Yaskawa INFORM job: MALBEN4.JBI

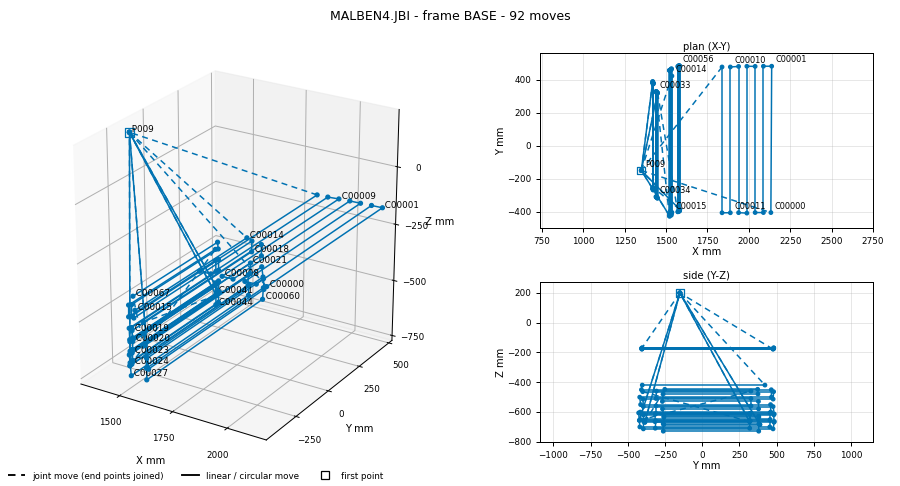
[picture p0: tool path of MALBEN4.JBI in frame BASE, 92 of 92 moves have a stored position in this frame; points joined in program order, loops and branches not executed]
/JOB
//NAME MALBEN4
//POS
///NPOS 86,0,86,1,0,1
///TOOL 0
///POSTYPE BASE
///RECTAN
///RCONF 1,0,0,1,1,0,0,0,0,0,0,0,0,0,0,0,0,0,0,0,0,0,0,0
C00000=2133.293,-404.385,-169.038,175.0001,4.9994,4.9985
///RCONF 1,0,0,0,0,0,0,0,0,0,0,0,0,0,0,0,0,0,0,0,0,0,0,0
C00001=2138.089,480.563,-169.043,175.0000,5.0000,5.0000
C00002=2088.089,480.435,-170.096,175.0000,5.0000,5.0000
C00003=2088.089,-404.293,-170.096,175.0000,5.0000,5.0000
C00004=2038.089,-404.161,-171.304,175.0000,5.0000,5.0000
C00005=2038.089,479.548,-171.304,175.0000,5.0000,5.0000
C00006=1988.089,480.242,-172.720,175.0000,5.0000,5.0000
C00007=1988.089,-407.599,-172.720,175.0000,5.0000,5.0000
C00008=1938.089,-404.906,-174.491,175.0000,5.0000,5.0000
C00009=1938.089,479.135,-174.491,175.0000,5.0000,5.0000
C00010=1888.089,475.934,-176.316,175.0000,5.0000,5.0000
C00011=1888.089,-405.530,-176.316,175.0000,5.0000,5.0000
C00012=1837.950,-405.573,-177.808,175.0000,5.0000,5.0000
C00013=1837.950,475.917,-177.808,175.0000,5.0000,5.0000
C00014=1534.901,421.478,-419.338,175.0000,-89.9999,5.0000
C00015=1534.901,-402.937,-419.338,175.0000,-89.9999,5.0000
C00016=1533.144,-408.647,-450.491,175.0000,-89.9999,5.0000
C00017=1533.144,464.153,-450.491,175.0000,-89.9999,5.0000
C00018=1531.375,464.936,-500.491,175.0000,-89.9999,5.0000
C00019=1531.375,-420.046,-500.491,175.0000,-89.9999,5.0000
C00020=1529.352,-413.942,-550.491,175.0000,-89.9999,5.0000
C00021=1529.352,459.233,-550.491,175.0000,-89.9999,5.0000
C00022=1526.912,460.521,-600.491,175.0000,-89.9999,5.0000
C00023=1526.912,-416.386,-600.491,175.0000,-89.9999,5.0000
C00024=1524.500,-416.295,-650.491,175.0000,-89.9999,5.0000
C00025=1524.500,456.784,-650.491,175.0000,-89.9999,5.0000
C00026=1522.504,454.310,-700.491,175.0000,-89.9999,5.0000
C00027=1522.504,-419.163,-700.491,175.0000,-89.9999,5.0000
C00028=1520.880,-427.203,-606.153,180.0000,-60.0000,0.0000
C00029=1520.880,455.493,-606.153,180.0000,-60.0000,0.0000
C00030=1519.374,455.436,-656.153,180.0000,-60.0000,0.0000
C00031=1519.374,-422.503,-656.153,180.0000,-60.0000,0.0000
C00032=1519.374,-422.503,-656.153,180.0000,-60.0000,0.0000
C00033=1438.715,327.474,-459.345,175.0000,-89.9999,5.0000
C00034=1438.715,-307.755,-459.345,175.0000,-89.9999,5.0000
C00035=1439.798,-310.872,-509.345,175.0000,-89.9999,5.0000
C00036=1439.798,327.369,-509.345,175.0000,-89.9999,5.0000
C00037=1441.037,327.734,-559.345,175.0000,-89.9999,5.0000
C00038=1441.037,-310.730,-559.345,175.0000,-89.9999,5.0000
C00039=1442.396,-310.620,-609.345,175.0000,-89.9999,5.0000
C00040=1442.396,320.382,-609.345,175.0000,-89.9999,5.0000
C00041=1443.632,322.978,-659.345,175.0000,-89.9999,5.0000
C00042=1443.632,-311.906,-659.345,175.0000,-89.9999,5.0000
C00043=1445.183,-315.667,-709.345,175.0000,-89.9999,5.0000
C00044=1445.183,319.105,-709.345,175.0000,-89.9999,5.0000
C00045=1446.831,319.750,-615.007,180.0000,-60.0000,0.0000
C00046=1446.831,-315.758,-615.007,180.0000,-60.0000,0.0000
C00047=1448.220,-317.504,-665.007,180.0000,-60.0000,0.0000
C00048=1448.220,318.562,-665.007,180.0000,-60.0000,0.0000
C00049=1448.220,318.562,-665.007,180.0000,-60.0000,0.0000
C00050=1570.356,-399.922,-463.648,175.0000,-89.9999,5.0000
C00051=1570.356,479.704,-463.648,175.0000,-89.9999,5.0000
C00052=1572.586,476.504,-513.648,175.0000,-89.9999,5.0000
C00053=1572.586,-398.280,-513.648,175.0000,-89.9999,5.0000
C00054=1574.691,-395.744,-563.648,175.0000,-89.9999,5.0000
C00055=1574.691,476.324,-563.648,175.0000,-89.9999,5.0000
C00056=1576.436,484.068,-613.648,175.0000,-89.9999,5.0000
C00057=1576.436,-394.544,-613.648,175.0000,-89.9999,5.0000
C00058=1578.039,-393.977,-663.648,175.0000,-89.9999,5.0000
C00059=1578.039,484.690,-663.648,175.0000,-89.9999,5.0000
C00060=1579.649,475.998,-713.648,175.0000,-89.9999,5.0000
C00061=1579.649,-395.540,-713.648,175.0000,-89.9999,5.0000
C00062=1580.841,-394.570,-619.310,180.0000,-60.0000,0.0000
C00063=1580.841,480.898,-619.310,180.0000,-60.0000,0.0000
C00064=1582.269,482.315,-669.310,180.0000,-60.0000,0.0000
C00065=1582.269,-385.635,-669.310,180.0000,-60.0000,0.0000
C00066=1582.269,-385.635,-669.310,180.0000,-60.0000,0.0000
C00067=1420.964,-251.559,-447.665,175.0000,-89.9999,5.0000
C00068=1420.964,372.604,-447.665,175.0000,-89.9999,5.0000
C00069=1422.373,374.697,-479.185,175.0000,-89.9999,5.0000
C00070=1422.373,-263.019,-479.185,175.0000,-89.9999,5.0000
C00071=1421.975,-267.696,-529.185,175.0000,-89.9999,5.0000
C00072=1421.975,377.834,-529.185,175.0000,-89.9999,5.0000
C00073=1421.594,378.934,-579.185,175.0000,-89.9999,5.0000
C00074=1421.594,-266.992,-579.185,175.0000,-89.9999,5.0000
C00075=1420.418,-258.080,-629.185,175.0000,-89.9999,5.0000
C00076=1420.418,379.690,-629.185,175.0000,-89.9999,5.0000
C00077=1419.981,380.884,-679.185,175.0000,-89.9999,5.0000
C00078=1419.981,-262.435,-679.185,175.0000,-89.9999,5.0000
C00079=1419.737,-261.680,-729.185,175.0000,-89.9999,5.0000
C00080=1419.737,379.769,-729.185,175.0000,-89.9999,5.0000
C00081=1419.270,380.316,-634.847,180.0000,-60.0000,0.0000
C00082=1419.270,-257.794,-634.847,180.0000,-60.0000,0.0000
C00083=1418.737,-258.418,-684.847,180.0000,-60.0000,0.0000
C00084=1418.737,387.426,-684.847,180.0000,-60.0000,0.0000
C00085=1418.737,387.426,-684.847,180.0000,-60.0000,0.0000
///POSTYPE PULSE
///PULSE
EC00000=0
EC00001=0
EC00002=0
EC00003=0
EC00004=0
EC00005=0
EC00006=0
EC00007=0
EC00008=0
EC00009=0
EC00010=0
EC00011=0
EC00012=0
EC00013=0
EC00014=0
EC00015=0
EC00016=0
EC00017=0
EC00018=0
EC00019=0
EC00020=0
EC00021=0
EC00022=0
EC00023=0
EC00024=0
EC00025=0
EC00026=0
EC00027=0
EC00028=0
EC00029=0
EC00030=0
EC00031=0
EC00032=92160
EC00033=92160
EC00034=92160
EC00035=92160
EC00036=92160
EC00037=92160
EC00038=92160
EC00039=92160
EC00040=92160
EC00041=92160
EC00042=92160
EC00043=92160
EC00044=92160
EC00045=92160
EC00046=92160
EC00047=92160
EC00048=92160
EC00049=184320
EC00050=184320
EC00051=184320
EC00052=184320
EC00053=184320
EC00054=184320
EC00055=184320
EC00056=184320
EC00057=184320
EC00058=184320
EC00059=184320
EC00060=184320
EC00061=184320
EC00062=184320
EC00063=184320
EC00064=184320
EC00065=184320
EC00066=276480
EC00067=276480
EC00068=276480
EC00069=276480
EC00070=276480
EC00071=276480
EC00072=276480
EC00073=276480
EC00074=276480
EC00075=276480
EC00076=276480
EC00077=276480
EC00078=276480
EC00079=276480
EC00080=276480
EC00081=276480
EC00082=276480
EC00083=276480
EC00084=276480
EC00085=368640
///POSTYPE BASE
///RECTAN
P00009=1350.000,-150.000,200.000,-180.0000,-45.0000,0.0000
///POSTYPE PULSE
///PULSE
EX00000=0
//INST
///DATE 2023/06/22 12:19
///ATTR SC,RW,RJ
////FRAME BASE
///GROUP1 RB1,ST1
NOP
MOVJ P009 EX000 VJ=15.00
MOVJ C00000 EC00000 VJ=15.00
MOVL C00001 EC00001 V=300.0
MOVL C00002 EC00002 V=300.0
MOVL C00003 EC00003 V=300.0
MOVL C00004 EC00004 V=300.0
MOVL C00005 EC00005 V=300.0
MOVL C00006 EC00006 V=300.0
MOVL C00007 EC00007 V=300.0
MOVL C00008 EC00008 V=300.0
MOVL C00009 EC00009 V=300.0
MOVL C00010 EC00010 V=300.0
MOVL C00011 EC00011 V=300.0
MOVL C00012 EC00012 V=300.0
MOVL C00013 EC00013 V=300.0
MOVJ P009 VJ=15.00
MOVJ C00014 EC00014 VJ=15.00
MOVL C00015 EC00015 V=300.0
MOVL C00016 EC00016 V=300.0
MOVL C00017 EC00017 V=300.0
MOVL C00018 EC00018 V=300.0
MOVL C00019 EC00019 V=300.0
MOVL C00020 EC00020 V=300.0
MOVL C00021 EC00021 V=300.0
MOVL C00022 EC00022 V=300.0
MOVL C00023 EC00023 V=300.0
MOVL C00024 EC00024 V=300.0
MOVL C00025 EC00025 V=300.0
MOVL C00026 EC00026 V=300.0
MOVL C00027 EC00027 V=300.0
MOVL C00028 EC00028 V=300.0
MOVL C00029 EC00029 V=300.0
MOVL C00030 EC00030 V=300.0
MOVL C00031 EC00031 V=300.0
MOVJ P009 VJ=15.00
MOVL C00032 EC00032 V=300.0
MOVJ C00033 EC00033 VJ=15.00
MOVL C00034 EC00034 V=300.0
MOVL C00035 EC00035 V=300.0
MOVL C00036 EC00036 V=300.0
MOVL C00037 EC00037 V=300.0
MOVL C00038 EC00038 V=300.0
MOVL C00039 EC00039 V=300.0
MOVL C00040 EC00040 V=300.0
MOVL C00041 EC00041 V=300.0
MOVL C00042 EC00042 V=300.0
MOVL C00043 EC00043 V=300.0
MOVL C00044 EC00044 V=300.0
MOVL C00045 EC00045 V=300.0
MOVL C00046 EC00046 V=300.0
MOVL C00047 EC00047 V=300.0
MOVL C00048 EC00048 V=300.0
MOVJ P009 VJ=15.00
MOVL C00049 EC00049 V=300.0
MOVJ C00050 EC00050 VJ=15.00
MOVL C00051 EC00051 V=300.0
MOVL C00052 EC00052 V=300.0
MOVL C00053 EC00053 V=300.0
MOVL C00054 EC00054 V=300.0
MOVL C00055 EC00055 V=300.0
MOVL C00056 EC00056 V=300.0
MOVL C00057 EC00057 V=300.0
MOVL C00058 EC00058 V=300.0
MOVL C00059 EC00059 V=300.0
MOVL C00060 EC00060 V=300.0
MOVL C00061 EC00061 V=300.0
MOVL C00062 EC00062 V=300.0
MOVL C00063 EC00063 V=300.0
MOVL C00064 EC00064 V=300.0
MOVL C00065 EC00065 V=300.0
MOVJ P009 VJ=15.00
MOVL C00066 EC00066 V=300.0
MOVJ C00067 EC00067 VJ=15.00
MOVL C00068 EC00068 V=300.0
MOVL C00069 EC00069 V=300.0
MOVL C00070 EC00070 V=300.0
MOVL C00071 EC00071 V=300.0
MOVL C00072 EC00072 V=300.0
MOVL C00073 EC00073 V=300.0
MOVL C00074 EC00074 V=300.0
MOVL C00075 EC00075 V=300.0
MOVL C00076 EC00076 V=300.0
MOVL C00077 EC00077 V=300.0
MOVL C00078 EC00078 V=300.0
MOVL C00079 EC00079 V=300.0
MOVL C00080 EC00080 V=300.0
MOVL C00081 EC00081 V=300.0
MOVL C00082 EC00082 V=300.0
MOVL C00083 EC00083 V=300.0
MOVL C00084 EC00084 V=300.0
MOVJ P009 VJ=15.00
MOVL C00085 EC00085 V=300.0
END
